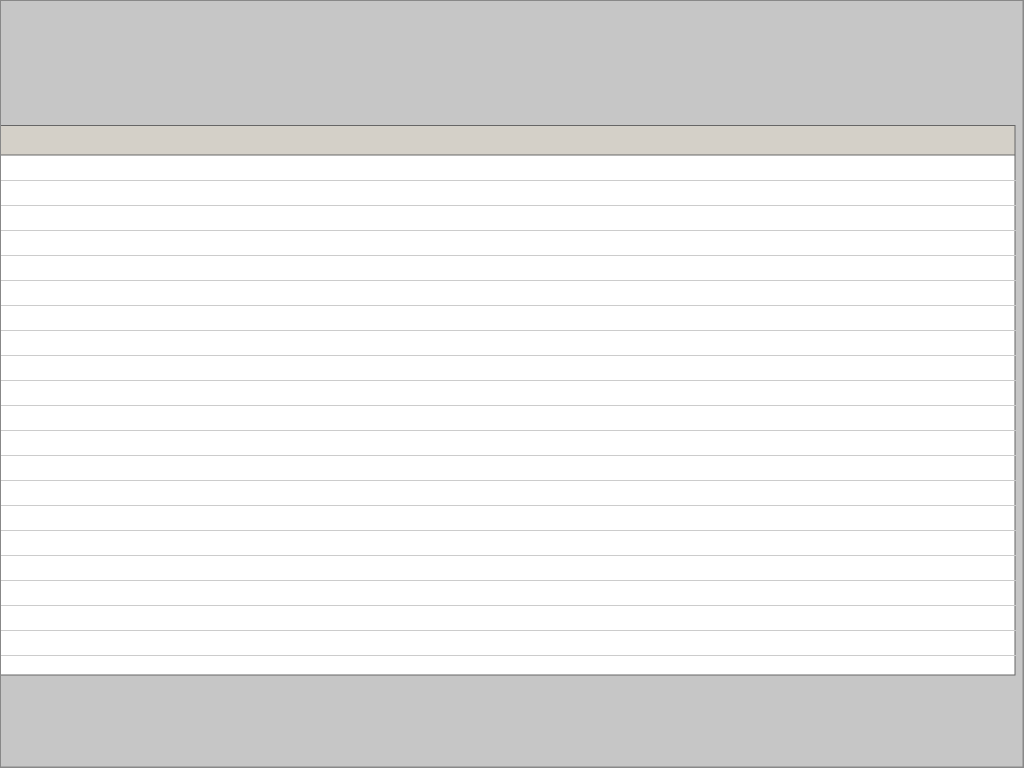
VISUALIZATION Msg_021_AlarmsView  // 1024x768
    Frame (0,0 1024x768)
        shows Tmp_000_Template(header := gHMIData.hmiHeader)
    Table (0,125 1015x550), data array: GlobalMessages.gHMIAlarmView.msgArry
        p3854506369: GlobalMessages.gHMIAlarmView.msgArry[INDEX].timeRaised
        p1892666644: GlobalMessages.gHMIAlarmView.msgArry[INDEX].text
        p338671338: GlobalMessages.gHMIAlarmView.msgArry[INDEX].timeResolved
        p2170511999: GlobalMessages.gHMIAlarmView.msgArry[INDEX].source
        p2232123230: Time Raised
        p511219082: Message Text
        p1755163831: Time Resolved
        p4092479075: Location
        Columns.Column.[0].Template: GlobalMessages.gHMIAlarmView.msgArryStyle[INDEX].isColoured; GlobalMessages.gHMIAlarmView.msgArryStyle[INDEX].colourToApply
        Columns.Column.[1].Template: GlobalMessages.gHMIAlarmView.msgArryStyle[INDEX].isColoured; GlobalMessages.gHMIAlarmView.msgArryStyle[INDEX].colourToApply
        Columns.Column.[2].Template: GlobalMessages.gHMIAlarmView.msgArryStyle[INDEX].isColoured; GlobalMessages.gHMIAlarmView.msgArryStyle[INDEX].colourToApply
        Columns.Column.[3].Template: GlobalMessages.gHMIAlarmView.msgArryStyle[INDEX].isColoured; GlobalMessages.gHMIAlarmView.msgArryStyle[INDEX].colourToApply
END_VISUALIZATION

(* stored: Version 1.1.0.1, ProductVersion 3.1.4024.12
   Visu Msg_021_AlarmsView: Id {f0caa955-e950-4402-b6fa-6d4c00190f56} *)
